FUNCTION_BLOCK ep7xxxBasicAxis_FB EXTENDS BeckHoffBasicAxis_FB
VAR_INPUT
	rDriveEnable: 	REFERENCE TO BOOL; // Reference to external drive enable signal
END_VAR
VAR_OUTPUT
END_VAR
VAR
	
END_VAR


AxisCtrlPtr^.Input.Parameter.Drive.eDriveType	:= enumDriveType.eEP70xx;
AxisCtrlPtr^.Input.Parameter.Drive.VendorNameID	:= eVendorNameID.Beckhoff;

SUPER^(AxisRef:=AxisRef);

IF __ISVALIDREF(rDriveEnable) THEN
	AxisCtrlPtr^.Output.Status.DriveEnable	:= rDriveEnable;
ELSE
	AxisCtrlPtr^.Output.Status.DriveEnable	:= TRUE;
END_IF

END_FUNCTION_BLOCK

(* stored: Version 1.1.0.1, ProductVersion 3.1.4024.3
   POU ep7xxxBasicAxis_FB: Id {5e591c83-a41e-4c28-9fcd-59c96779611c}, SpecialFunc None *)
